(* PLC project Sin nombre, Desconocido Sin nombre 1 *)
(* stored: creationDateTime 2023-02-22T01:16:49, modificationDateTime 2023-02-22T01:19:17 *)

PROGRAM Example_1
  VAR
    PushButton AT %IX0.0 : BOOL;  (* Ejemplo de entrada tipo Booleano *)
    Salida AT %QX0.0 : BOOL;  (* Ejemplo de salida tipo Booleano *)
  END_VAR

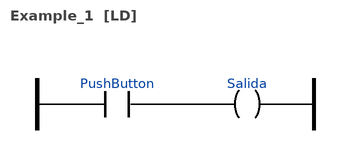
(* LD diagram, written out as Structured Text *)
Salida := PushButton;
END_PROGRAM

CONFIGURATION Config0
  RESOURCE Res0 ON PLC
    TASK task0(INTERVAL := T#20ms, PRIORITY := 0);
    PROGRAM instance0 WITH task0 : Example_1;
  END_RESOURCE
END_CONFIGURATION
